PROGRAM MAIN
VAR
	Ablauf: FB_Ablauf;
	Betriebsarten: FB_Betriebsarten;
END_VAR

Ablauf(stAnlagenzustand := Betriebsarten.stAnlagenzustand);
Betriebsarten();

END_PROGRAM

(* stored: Version 1.1.0.1
   POU MAIN: Id {d461958c-9aaf-4c1a-b6af-a9b25b2a3433}, SpecialFunc None *)
